// TIA Portal V20 export
TYPE "typeSequenceControlNodeJobInterfaceMonitoring"
// stored: Namespace Unit1.Em1
   STRUCT
      busyRewind { ExternalWritable := 'False'} : Bool;
      busyLinkChg { ExternalWritable := 'False'} : Bool;
      doneRewind { ExternalWritable := 'False'} : Bool;
      doneLinkChg { ExternalWritable := 'False'} : Bool;
   END_STRUCT;
END_TYPE
